// TIA Portal V16 export
// export: Created 2024-05-10T06:46:39.4006194Z, ExportSetting WithDefaults, DisplayName Totally Integrated Automation Portal, DisplayVersion V16, DisplayName TIA Portal Version Control Interface, DisplayVersion V16, DisplayName TIA Portal Openness, DisplayVersion V16, DisplayName STEP 7 Professional, DisplayVersion V16, DisplayName STEP 7 Safety, DisplayVersion V16, DisplayName WinCC Professional, DisplayVersion V16
ORGANIZATION_BLOCK "Main"   // OB1, LAD, ProgramCycle
TITLE = "Main Program Sweep (Cycle)"
{ S7_Optimized_Access := 'TRUE' }
VERSION : 0.1
// stored: AutoNumber true, IsIECCheckEnabled false, SetENOAutomatically false
   VAR_INPUT
      Initial_Call : Bool;   // Initial call of this OB
      Remanence : Bool;   // =True, if remanent data are available
   END_VAR
   VAR_TEMP
      PLC_Date_Read : DTL;
      PLC_DateState_R : Int;
      PLC_Date_Write : DTL;
      PLC_DateState_W : Int;
      M_pulse : Array[1..10] of Bool;
      W_SecCont : Array[1..5] of Int;
   END_VAR
   VAR_TEMP   // added for the SCL form of the ladder/FBD networks
      _w1 : Bool;
      _w2 : Bool;
   END_VAR
BEGIN

REGION Network 1: FB调用
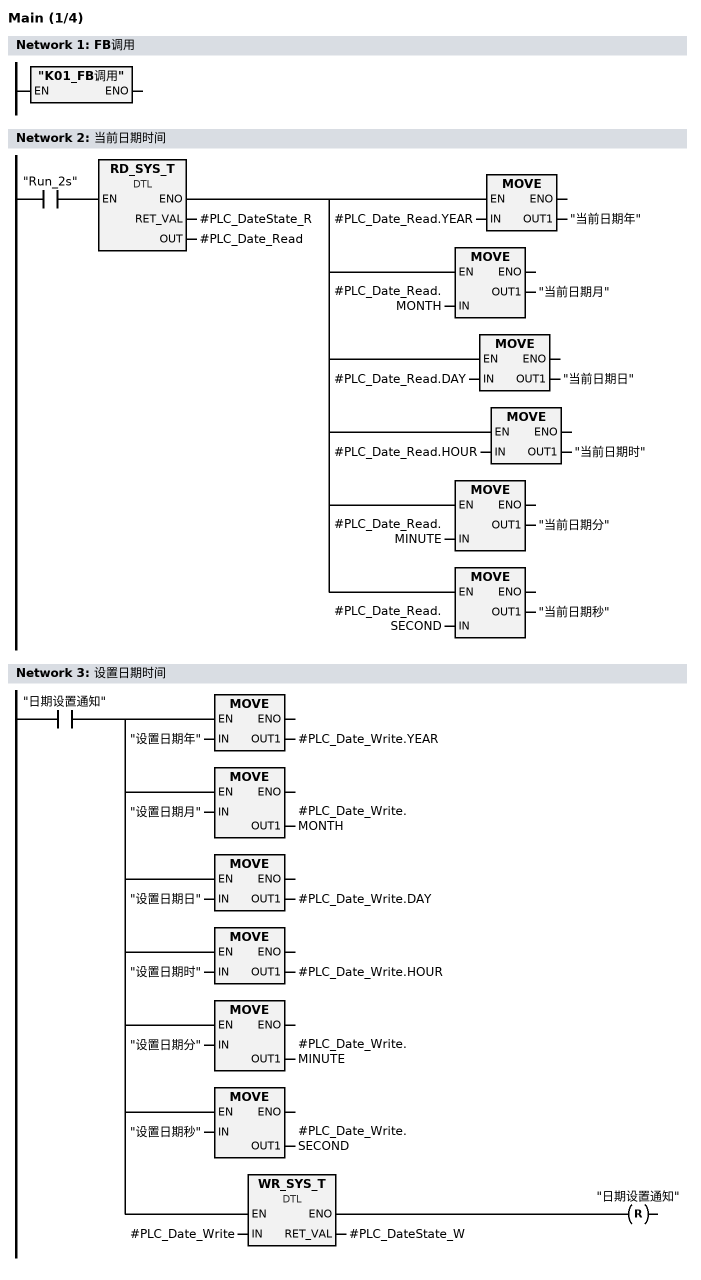
   RUNG wire#powerrail
      "K01_FB调用"()
   END_RUNG
   // the same network as SCL:
   "K01_FB调用"();
END_REGION

REGION Network 2: 当前日期时间
   RUNG wire#powerrail
      Contact( "Run_2s" )
      { S7_Templates := "date_type := DTL" } RD_SYS_T(RET_VAL => #PLC_DateState_R, OUT => #PLC_Date_Read)
      wire#w1
      Move(in := #PLC_Date_Read.YEAR, out1 => "当前日期年")
   END_RUNG
   RUNG wire#w1
      Move(in := #PLC_Date_Read.MONTH, out1 => "当前日期月")
   END_RUNG
   RUNG wire#w1
      Move(in := #PLC_Date_Read.DAY, out1 => "当前日期日")
   END_RUNG
   RUNG wire#w1
      Move(in := #PLC_Date_Read.HOUR, out1 => "当前日期时")
   END_RUNG
   RUNG wire#w1
      Move(in := #PLC_Date_Read.MINUTE, out1 => "当前日期分")
   END_RUNG
   RUNG wire#w1
      Move(in := #PLC_Date_Read.SECOND, out1 => "当前日期秒")
   END_RUNG
   // the same network as SCL:
   #PLC_DateState_R := RD_SYS_T(EN := "Run_2s", OUT => #PLC_Date_Read, ENO => #_w1);
   IF #_w1 THEN
       "当前日期年" := #PLC_Date_Read.YEAR;
       "当前日期月" := #PLC_Date_Read.MONTH;
       "当前日期日" := #PLC_Date_Read.DAY;
       "当前日期时" := #PLC_Date_Read.HOUR;
       "当前日期分" := #PLC_Date_Read.MINUTE;
       "当前日期秒" := #PLC_Date_Read.SECOND;
   END_IF;
END_REGION

REGION Network 3: 设置日期时间
   RUNG wire#powerrail
      Contact( "日期设置通知" )
      wire#w1
      Move(in := "设置日期年", out1 => #PLC_Date_Write.YEAR)
   END_RUNG
   RUNG wire#w1
      Move(in := "设置日期月", out1 => #PLC_Date_Write.MONTH)
   END_RUNG
   RUNG wire#w1
      Move(in := "设置日期日", out1 => #PLC_Date_Write.DAY)
   END_RUNG
   RUNG wire#w1
      Move(in := "设置日期时", out1 => #PLC_Date_Write.HOUR)
   END_RUNG
   RUNG wire#w1
      Move(in := "设置日期分", out1 => #PLC_Date_Write.MINUTE)
   END_RUNG
   RUNG wire#w1
      Move(in := "设置日期秒", out1 => #PLC_Date_Write.SECOND)
   END_RUNG
   RUNG wire#w1
      { S7_Templates := "date_type := DTL" } WR_SYS_T(IN := #PLC_Date_Write, RET_VAL => #PLC_DateState_W)
      R_Coil( "日期设置通知" )
   END_RUNG
   // the same network as SCL:
   IF "日期设置通知" THEN
       #PLC_Date_Write.YEAR := "设置日期年";
       #PLC_Date_Write.MONTH := "设置日期月";
       #PLC_Date_Write.DAY := "设置日期日";
       #PLC_Date_Write.HOUR := "设置日期时";
       #PLC_Date_Write.MINUTE := "设置日期分";
       #PLC_Date_Write.SECOND := "设置日期秒";
   END_IF;
   #PLC_DateState_W := WR_SYS_T(EN := "日期设置通知", IN := #PLC_Date_Write, ENO => #_w1);
   IF #_w1 THEN "日期设置通知" := FALSE; END_IF;
END_REGION

REGION Network 4: 开机日期时间
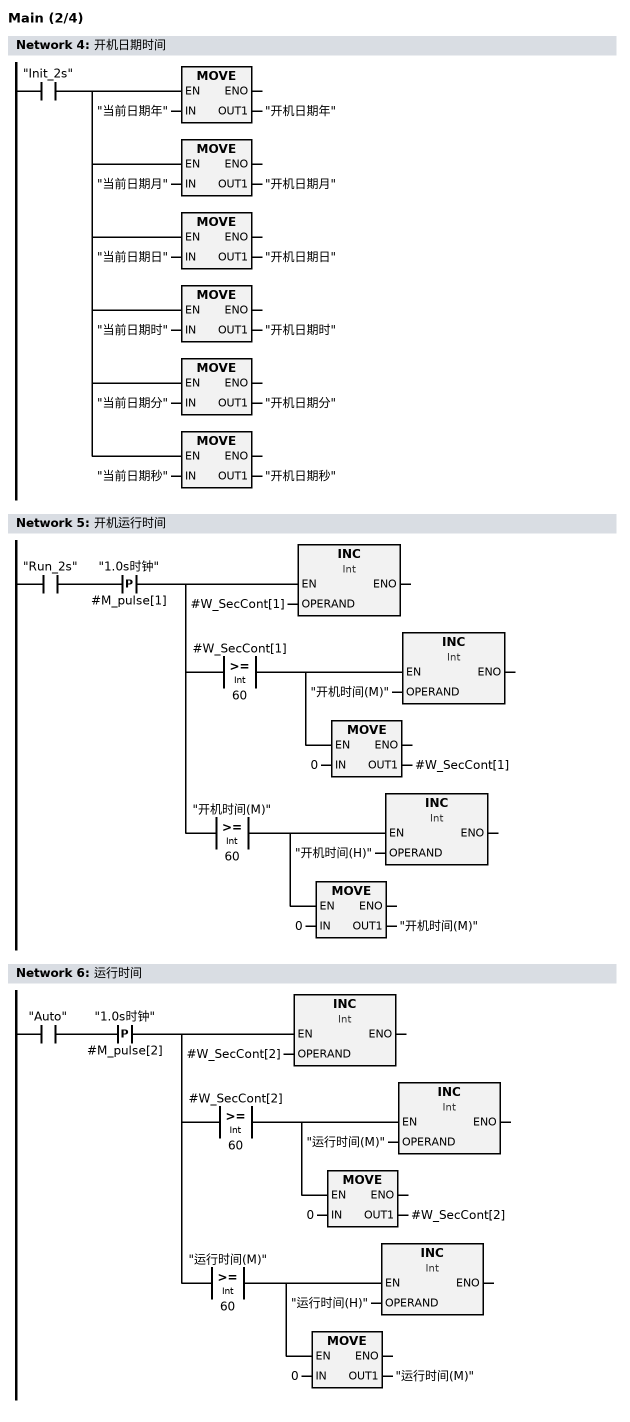
   RUNG wire#powerrail
      Contact( "Init_2s" )
      wire#w1
      Move(in := "当前日期年", out1 => "开机日期年")
   END_RUNG
   RUNG wire#w1
      Move(in := "当前日期月", out1 => "开机日期月")
   END_RUNG
   RUNG wire#w1
      Move(in := "当前日期日", out1 => "开机日期日")
   END_RUNG
   RUNG wire#w1
      Move(in := "当前日期时", out1 => "开机日期时")
   END_RUNG
   RUNG wire#w1
      Move(in := "当前日期分", out1 => "开机日期分")
   END_RUNG
   RUNG wire#w1
      Move(in := "当前日期秒", out1 => "开机日期秒")
   END_RUNG
   // the same network as SCL:
   IF "Init_2s" THEN
       "开机日期年" := "当前日期年";
       "开机日期月" := "当前日期月";
       "开机日期日" := "当前日期日";
       "开机日期时" := "当前日期时";
       "开机日期分" := "当前日期分";
       "开机日期秒" := "当前日期秒";
   END_IF;
END_REGION

REGION Network 5: 开机运行时间
   RUNG wire#powerrail
      Contact( "Run_2s" )
      P_Contact(operand := "1.0s时钟", bit := #M_pulse[1])
      wire#w1
      { S7_Templates := "DestType := Int" } Inc( #W_SecCont[1] )
   END_RUNG
   RUNG wire#w1
      { S7_Templates := "SrcType := Int" } GE_Contact(in1 := #W_SecCont[1], in2 := 60)
      wire#w2
      { S7_Templates := "DestType := Int" } Inc( "开机时间(M)" )
   END_RUNG
   RUNG wire#w2
      Move(in := 0, out1 => #W_SecCont[1])
   END_RUNG
   RUNG wire#w1
      { S7_Templates := "SrcType := Int" } GE_Contact(in1 := "开机时间(M)", in2 := 60)
      wire#w3
      { S7_Templates := "DestType := Int" } Inc( "开机时间(H)" )
   END_RUNG
   RUNG wire#w3
      Move(in := 0, out1 => "开机时间(M)")
   END_RUNG
   // the same network as SCL:
   #_w1 := "Run_2s" AND "1.0s时钟" AND NOT #M_pulse[1];   // rising edge of "1.0s时钟"
   #M_pulse[1] := "1.0s时钟";
   IF #_w1 THEN #W_SecCont[1] := #W_SecCont[1] + 1; END_IF;
   IF #_w1 AND (#W_SecCont[1] >= 60) THEN
       "开机时间(M)" := "开机时间(M)" + 1;
       #W_SecCont[1] := 0;
   END_IF;
   IF #_w1 AND ("开机时间(M)" >= 60) THEN
       "开机时间(H)" := "开机时间(H)" + 1;
       "开机时间(M)" := 0;
   END_IF;
END_REGION

REGION Network 6: 运行时间
   RUNG wire#powerrail
      Contact( "Auto" )
      P_Contact(operand := "1.0s时钟", bit := #M_pulse[2])
      wire#w1
      { S7_Templates := "DestType := Int" } Inc( #W_SecCont[2] )
   END_RUNG
   RUNG wire#w1
      { S7_Templates := "SrcType := Int" } GE_Contact(in1 := #W_SecCont[2], in2 := 60)
      wire#w2
      { S7_Templates := "DestType := Int" } Inc( "运行时间(M)" )
   END_RUNG
   RUNG wire#w2
      Move(in := 0, out1 => #W_SecCont[2])
   END_RUNG
   RUNG wire#w1
      { S7_Templates := "SrcType := Int" } GE_Contact(in1 := "运行时间(M)", in2 := 60)
      wire#w3
      { S7_Templates := "DestType := Int" } Inc( "运行时间(H)" )
   END_RUNG
   RUNG wire#w3
      Move(in := 0, out1 => "运行时间(M)")
   END_RUNG
   // the same network as SCL:
   #_w1 := "Auto" AND "1.0s时钟" AND NOT #M_pulse[2];   // rising edge of "1.0s时钟"
   #M_pulse[2] := "1.0s时钟";
   IF #_w1 THEN #W_SecCont[2] := #W_SecCont[2] + 1; END_IF;
   IF #_w1 AND (#W_SecCont[2] >= 60) THEN
       "运行时间(M)" := "运行时间(M)" + 1;
       #W_SecCont[2] := 0;
   END_IF;
   IF #_w1 AND ("运行时间(M)" >= 60) THEN
       "运行时间(H)" := "运行时间(H)" + 1;
       "运行时间(M)" := 0;
   END_IF;
END_REGION

REGION Network 7: 停止时间
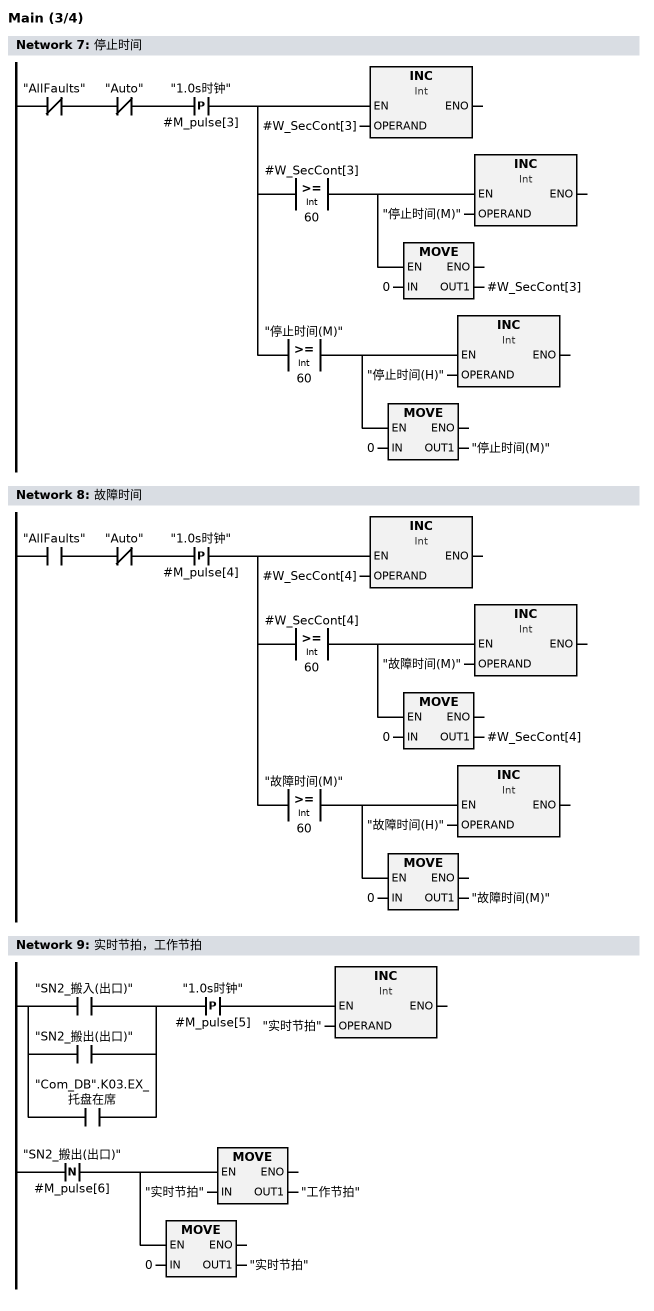
   RUNG wire#powerrail
      I_Contact( "AllFaults" )
      I_Contact( "Auto" )
      P_Contact(operand := "1.0s时钟", bit := #M_pulse[3])
      wire#w1
      { S7_Templates := "DestType := Int" } Inc( #W_SecCont[3] )
   END_RUNG
   RUNG wire#w1
      { S7_Templates := "SrcType := Int" } GE_Contact(in1 := #W_SecCont[3], in2 := 60)
      wire#w2
      { S7_Templates := "DestType := Int" } Inc( "停止时间(M)" )
   END_RUNG
   RUNG wire#w2
      Move(in := 0, out1 => #W_SecCont[3])
   END_RUNG
   RUNG wire#w1
      { S7_Templates := "SrcType := Int" } GE_Contact(in1 := "停止时间(M)", in2 := 60)
      wire#w3
      { S7_Templates := "DestType := Int" } Inc( "停止时间(H)" )
   END_RUNG
   RUNG wire#w3
      Move(in := 0, out1 => "停止时间(M)")
   END_RUNG
   // the same network as SCL:
   #_w1 := NOT "AllFaults" AND NOT "Auto" AND "1.0s时钟" AND NOT #M_pulse[3];   // rising edge of "1.0s时钟"
   #M_pulse[3] := "1.0s时钟";
   IF #_w1 THEN #W_SecCont[3] := #W_SecCont[3] + 1; END_IF;
   IF #_w1 AND (#W_SecCont[3] >= 60) THEN
       "停止时间(M)" := "停止时间(M)" + 1;
       #W_SecCont[3] := 0;
   END_IF;
   IF #_w1 AND ("停止时间(M)" >= 60) THEN
       "停止时间(H)" := "停止时间(H)" + 1;
       "停止时间(M)" := 0;
   END_IF;
END_REGION

REGION Network 8: 故障时间
   RUNG wire#powerrail
      Contact( "AllFaults" )
      I_Contact( "Auto" )
      P_Contact(operand := "1.0s时钟", bit := #M_pulse[4])
      wire#w1
      { S7_Templates := "DestType := Int" } Inc( #W_SecCont[4] )
   END_RUNG
   RUNG wire#w1
      { S7_Templates := "SrcType := Int" } GE_Contact(in1 := #W_SecCont[4], in2 := 60)
      wire#w2
      { S7_Templates := "DestType := Int" } Inc( "故障时间(M)" )
   END_RUNG
   RUNG wire#w2
      Move(in := 0, out1 => #W_SecCont[4])
   END_RUNG
   RUNG wire#w1
      { S7_Templates := "SrcType := Int" } GE_Contact(in1 := "故障时间(M)", in2 := 60)
      wire#w3
      { S7_Templates := "DestType := Int" } Inc( "故障时间(H)" )
   END_RUNG
   RUNG wire#w3
      Move(in := 0, out1 => "故障时间(M)")
   END_RUNG
   // the same network as SCL:
   #_w1 := "AllFaults" AND NOT "Auto" AND "1.0s时钟" AND NOT #M_pulse[4];   // rising edge of "1.0s时钟"
   #M_pulse[4] := "1.0s时钟";
   IF #_w1 THEN #W_SecCont[4] := #W_SecCont[4] + 1; END_IF;
   IF #_w1 AND (#W_SecCont[4] >= 60) THEN
       "故障时间(M)" := "故障时间(M)" + 1;
       #W_SecCont[4] := 0;
   END_IF;
   IF #_w1 AND ("故障时间(M)" >= 60) THEN
       "故障时间(H)" := "故障时间(H)" + 1;
       "故障时间(M)" := 0;
   END_IF;
END_REGION

REGION Network 9: 实时节拍，工作节拍
   RUNG wire#powerrail
      Contact( "SN2_搬入(出口)" )
      wire#w1
      P_Contact(operand := "1.0s时钟", bit := #M_pulse[5])
      { S7_Templates := "DestType := Int" } Inc( "实时节拍" )
   END_RUNG
   RUNG wire#powerrail
      Contact( "SN2_搬出(出口)" )
   END_RUNG wire#w1
   RUNG wire#powerrail
      Contact( "Com_DB".K03.EX_托盘在席 )
   END_RUNG wire#w1
   RUNG wire#powerrail
      N_Contact(operand := "SN2_搬出(出口)", bit := #M_pulse[6])
      wire#w2
      Move(in := "实时节拍", out1 => "工作节拍")
   END_RUNG
   RUNG wire#w2
      Move(in := 0, out1 => "实时节拍")
   END_RUNG
   // the same network as SCL:
   #_w1 := ("SN2_搬入(出口)" OR "SN2_搬出(出口)" OR "Com_DB".K03.EX_托盘在席) AND "1.0s时钟" AND NOT #M_pulse[5];   // rising edge of "1.0s时钟"
   #M_pulse[5] := "1.0s时钟";
   IF #_w1 THEN "实时节拍" := "实时节拍" + 1; END_IF;
   #_w2 := NOT "SN2_搬出(出口)" AND #M_pulse[6];   // falling edge of "SN2_搬出(出口)"
   #M_pulse[6] := "SN2_搬出(出口)";
   IF #_w2 THEN
       "工作节拍" := "实时节拍";
       "实时节拍" := 0;
   END_IF;
END_REGION

REGION Network 10: 生产数量. 累计数量
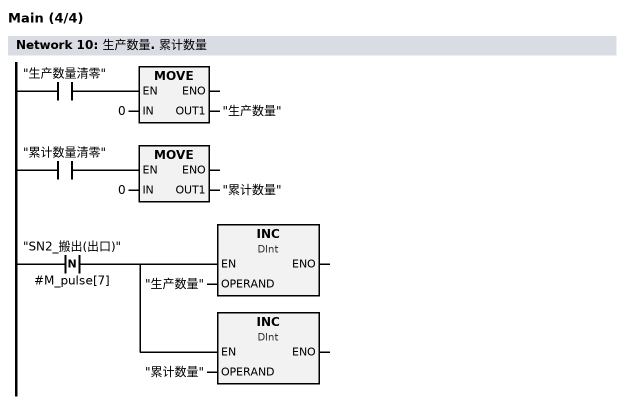
   RUNG wire#powerrail
      Contact( "生产数量清零" )
      Move(in := 0, out1 => "生产数量")
   END_RUNG
   RUNG wire#powerrail
      Contact( "累计数量清零" )
      Move(in := 0, out1 => "累计数量")
   END_RUNG
   RUNG wire#powerrail
      N_Contact(operand := "SN2_搬出(出口)", bit := #M_pulse[7])
      wire#w1
      { S7_Templates := "DestType := DInt" } Inc( "生产数量" )
   END_RUNG
   RUNG wire#w1
      { S7_Templates := "DestType := DInt" } Inc( "累计数量" )
   END_RUNG
   // the same network as SCL:
   IF "生产数量清零" THEN "生产数量" := 0; END_IF;
   IF "累计数量清零" THEN "累计数量" := 0; END_IF;
   #_w1 := NOT "SN2_搬出(出口)" AND #M_pulse[7];   // falling edge of "SN2_搬出(出口)"
   #M_pulse[7] := "SN2_搬出(出口)";
   IF #_w1 THEN
       "生产数量" := "生产数量" + 1;
       "累计数量" := "累计数量" + 1;
   END_IF;
END_REGION

REGION Network 11: OK. NG数量
END_REGION

REGION Network 12 (SCL): 稼动率 合格率 PPM计算

   //稼动率计算
   IF ("运行时间(H)" + "运行时间(M)" > 0)
       AND("开机时间(H)" + "开机时间(M)" > 0)
       AND"1.0s时钟"=TRUE
   THEN
       "稼动率%"   :=REAL_TO_INT(("运行时间(H)" * 60 + "运行时间(M)")/("开机时间(H)" * 60 + "开机时间(M)"))*100 ;
   END_IF;
   // 合格率计算
   IF "OK数量">0
       AND "生产数量">0
       AND"1.0s时钟"=TRUE
   THEN
       "合格率%" := REAL_TO_INT("OK数量" / "生产数量")*100;
   END_IF;

   //PPM计算
   IF ("运行时间(H)" + "运行时间(M)" > 0)
       AND "1.0s时钟" = TRUE
   THEN
       "PPM" := REAL_TO_INT("生产数量" / ("运行时间(H)" * 60 + "运行时间(M)"));

   END_IF;
END_REGION

REGION Network 13 (SCL): 生产数据清除
   IF "Init_2s"=TRUE
   THEN
       #W_SecCont[1] := 0;
       "开机时间(H)" := 0;
       "开机时间(M)" := 0;
       #W_SecCont[2] := 0;
       "运行时间(H)" := 0;
       "运行时间(M)" := 0;
       #W_SecCont[3] := 0;
       "停止时间(H)" := 0;
       "停止时间(M)" := 0;
       #W_SecCont[4] := 0;
       "故障时间(H)" := 0;
       "故障时间(M)" := 0;
   //////////////
       "实时节拍"    := 0;
       "工作节拍"    := 0;
       "生产数量"    := 0;
       "OK数量"      := 0;
       "NG数量"      := 0;
       "稼动率%"     := 0;
       "合格率%"     := 0;
       "PPM"         := 0;

   END_IF;
END_REGION
END_ORGANIZATION_BLOCK
